INTERFACE I_SessionData EXTENDS I_Disposable

END_INTERFACE

(* stored: Version 1.1.0.1, ProductVersion 3.1.4024.12
   Itf I_SessionData: Id {d66f3fee-d6ee-0f12-1a9e-8bcdfb936cea} *)
